{attribute 'qualified_only'}
{attribute 'strict'}
{attribute 'to_string'}
TYPE E_CylinderCycle :
(
	startCheck 			:= 0,
	extendCylinder 		:= 100,
	verifyExtension 	:= 200,
	retractCylinder 	:= 300,
	verifyRetraction	:= 400,
	cylinderFault		:= 500
	
);
END_TYPE

(* stored: Version 1.1.0.1
   DUT E_CylinderCycle: Id {b190ce46-6b8e-41d1-945e-0e92ddccb84f} *)
